	DATA_BLOCK DB130
	TITLE =DBG030G  Bin high levels
	//COPYRIGHT:    (C) 2009  BUHLER AG, CH-9240 UZWIL, SWITZERLAND
	//
	//PRODUCT:      WinCoS_BIW01_09
	//
	//TITLE:        Bin high levels
	//                General group DB
	//                Allgemeine Gruppen-DB
	//
	//-------------------------------------------------------------------------
	//
	//IDENT:        AUTHOR:             DEPT:             DATE:
	//
	//P01_DB130.1.0 K.Renz              CSB41             13.Jan.2010
	//              1st Release
	//
	//-------------------------------------------------------------------------
	//
	//PURPOSE:
	//
	//MANUAL :
	//
	//RESTRICTIONS:
	//
	//-------------------------------------------------------------------------
	AUTHOR  : KR
	FAMILY  : USW
	NAME    : DBG030G
	VERSION : 00.00

	FB130
	BEGIN
	      #Gr.Par.ParObjectNo 	:=3000;
	      #Gr.Par.ParIdling      	:=0;
	      #Gr.Par.ParMgr	        :=False;
	      #Gr.Par.ParWgr	        :=False;
	      #Gr.Par.ParGgr	        :=True;
	      #Gr.Par.ParEmptyingTime 	:=0;
	      #Gr.Par.ParHornCode       :=99;
	END_DATA_BLOCK
